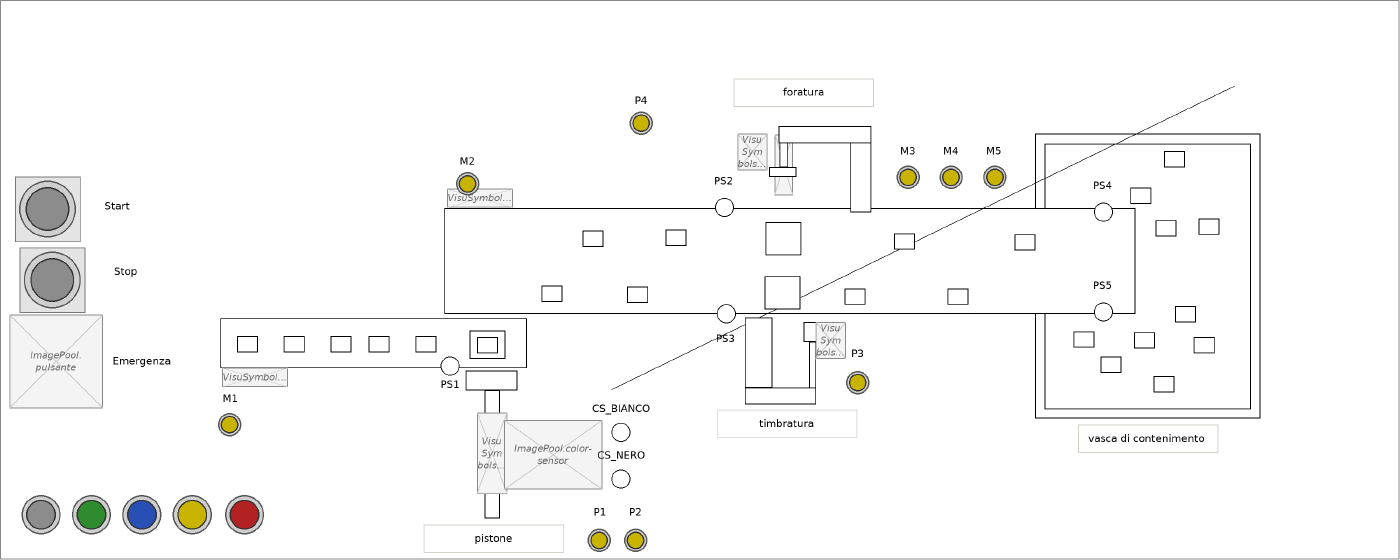
VISUALIZATION Visualization  // 1500x600
    PushSwitch (16,189 70x70), variable: GVL.PB1, behaviour: TAP, style: Switch-PushSwitch-Gray
    Label (98,206 55x30), "Start"
    PushSwitch (21,265 70x70), variable: GVL.PB2, behaviour: TAP, style: Switch-PushSwitch-Gray
    Label (102,276 65x30), "Stop"
    Label (107,372 90x30), "Emergenza"
    Lamp1 (20,527 48x49), variable: GVL.L1, style: Lamp-Lamp1-Gray
    Lamp1 (74,527 48x49), variable: GVL.L2, style: Lamp-Lamp1-Green
    Lamp1 (128,527 48x49), variable: GVL.L3, style: Lamp-Lamp1-Blue
    Lamp1 (182,527 48x49), variable: GVL.L4, style: Lamp-Lamp1-Yellow
    Lamp1 (238,527 48x49), variable: GVL.L5, style: Lamp-Lamp1-Red
    Image (10,337 100x100), image: ImagePool.pulsante
        OnMouseClick: toggle GVL.PBE
    Textfield (454,562 150x30), "pistone"
    Image (830,144 19x65), image: VisuSymbols.Symbols.ArrowBoldDown
    RoundedRectangle (1109,143 241x305)
    RoundedRectangle (1119,154 221x284)
    Rectangle (236,341 328x53)
    RoundedRectangle (476,223 740x113)
    Line (655,417) (1322,92)
    RoundedRectangle (499,397 55x21)
    Rectangle (519,418 16x137)
    Image (511,442 32x87), image: VisuSymbols.Symbols.DoubleArrow4
    Rectangle (254,360 22x17)
    Rectangle (304,360 22x17)
    Rectangle (354,360 22x17)
    Rectangle (395,360 22x17)
    Rectangle (624,247 22x17)
    Rectangle (713,246 22x17)
    Rectangle (445,360 22x17)
    Rectangle (580,306 22x17)
    Rectangle (672,307 22x17)
    Rectangle (905,309 22x17)
    Rectangle (1015,309 22x17)
    Rectangle (958,250 22x17)
    Rectangle (1087,251 22x17)
    Rectangle (1179,382 22x17)
    Rectangle (1279,361 22x17)
    Rectangle (1259,328 22x17)
    Rectangle (1215,356 22x17)
    Rectangle (1150,355 22x17)
    Rectangle (1236,403 22x17)
    Rectangle (1211,201 22x17)
    Rectangle (1247,162 22x17)
    Rectangle (1238,236 22x17)
    Rectangle (1284,234 22x17)
    Textfield (1155,455 150x30), "vasca di contenimento"
    RoundedRectangle (861,345 19x21)
    Rectangle (867,366 7x51)
    Rectangle (798,415 76x18)
    Rectangle (798,340 29x75)
    Image (874,345 32x39), image: VisuSymbols.Symbols.DoubleArrow4
    Textfield (768,439 150x30), "timbratura"
    Textfield (786,84 150x30), "foratura"
    Rectangle (911,152 22x75)
    RoundedRectangle (824,179 29x10)
    Rectangle (835,150 9x29)
    Rectangle (834,135 99x18)
    Image (790,143 32x39), image: VisuSymbols.Symbols.DoubleArrow4
    Image (479,202 70x20), image: VisuSymbols.Symbols.ArrowBoldRight
    Image (238,394 70x20), image: VisuSymbols.Symbols.ArrowBoldRight
    Rectangle (503,354 38x30)
    Rectangle (511,361 22x17)
    Rectangle (820,238 38x35)
    Rectangle (819,296 38x35)
    Label (205,412 84x30), "M1"
    Label (459,158 84x30), "M2"
    Lamp1 (232,440 28x30), variable: GVL.M1, style: Lamp-Lamp1-Yellow
    Lamp1 (487,182 28x30), variable: GVL.M2, style: Lamp-Lamp1-Yellow
    Ellipse (655,453 20x20), colour toggle: GVL.CS_BIANCO
        tap GVL.CS_BIANCO
    Label (623,432 85x12), "CS_BIANCO"
    Ellipse (472,382 20x20), colour toggle: GVL.PS1
        tap GVL.PS1
    Label (463,406 39x12), "PS1"
    Image (540,450 105x74), image: ImagePool.color-sensor
    Ellipse (655,503 20x20), colour toggle: GVL.CS_NERO
        tap GVL.CS_NERO
    Label (623,482 85x12), "CS_NERO"
    Label (601,534 84x30), "P1"
    Lamp1 (628,564 28x30), variable: GVL.P1, style: Lamp-Lamp1-Yellow
    Lamp1 (667,564 28x30), variable: GVL.P2, style: Lamp-Lamp1-Yellow
    Label (639,534 84x30), "P2"
    Label (756,188 39x12), "PS2"
    Ellipse (766,212 20x20), colour toggle: GVL.PS2
        tap GVL.PS2
    Label (758,357 39x12), "PS3"
    Ellipse (768,326 20x20), colour toggle: GVL.PS3
        tap GVL.PS3
    Label (645,93 84x30), "P4"
    Lamp1 (673,117 28x30), variable: GVL.P4, style: Lamp-Lamp1-Yellow
    Label (877,364 84x30), "P3"
    Lamp1 (905,395 28x30), variable: GVL.P3, style: Lamp-Lamp1-Yellow
    Lamp1 (959,175 28x30), variable: GVL.M3, style: Lamp-Lamp1-Yellow
    Label (931,147 84x30), "M3"
    Label (977,147 84x30), "M4"
    Lamp1 (1005,175 28x30), variable: GVL.M4, style: Lamp-Lamp1-Yellow
    Ellipse (1172,217 20x20), colour toggle: GVL.PS4
        tap GVL.PS4
    Label (1162,193 39x12), "PS4"
    Ellipse (1172,324 20x20), colour toggle: GVL.PS5
        tap GVL.PS5
    Label (1162,300 39x12), "PS5"
    Lamp1 (1052,175 28x30), variable: GVL.M5, style: Lamp-Lamp1-Yellow
    Label (1023,147 84x30), "M5"
END_VISUALIZATION

(* stored: Version 1.1.0.1, ProductVersion 3.1.4024.12
   Visu Visualization: Id {e3399594-b7fd-4589-9a49-3967da9e8e84} *)
